Fanuc KAREL source: kd00034.KL

-- PROVISIONAL review KL for V1013-1; original PC SHA256 9d27a4e0b62450b1ba18a6c292f281d3f4ea85650d065e6a9e6ef16e78b97f3e
-- Incomplete behavior may be omitted. Consult companion uncertainty JSON. Do not deploy.
PROGRAM KD00034
%NOLOCKGROUP
VAR
  I : INTEGER
  J : INTEGER
  B : BOOLEAN
  R : REAL
  S : STRING[80]
BEGIN
  -- UNRESOLVED_PC offsets 5-27; opcodes 9D,81,18,22,9D,12,22,9D,13,04
  -- UNRESOLVED_PC offsets 32-36; opcodes 7F
END KD00034
